REGION Network 162: Reset CV nước Bồn 3 khi không dosing
   RUNG wire#powerrail
      I_Contact( "PLC2_Step_Bon3_Dosing" )
      { S7_GenerateENO := "TRUE" } Move(in := 0.0, out1 => "CV3211_Nuoc_Bon3")
   END_RUNG
   // the same network as SCL:
   IF NOT "PLC2_Step_Bon3_Dosing" THEN "CV3211_Nuoc_Bon3" := 0.0; END_IF;
END_REGION

REGION Network 163: Reset CV nước Bồn 3 khi Stop hoặc Lỗi tổng PLC2
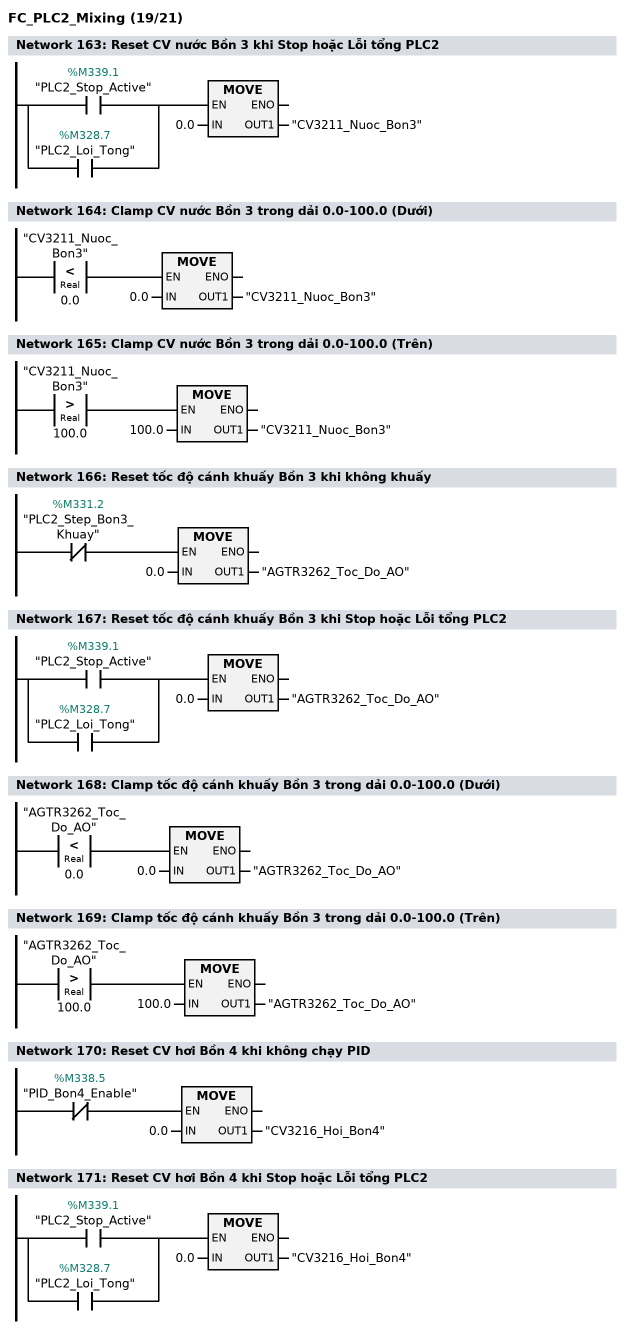
   RUNG wire#powerrail
      Contact( "PLC2_Stop_Active" )
      wire#w1
      { S7_GenerateENO := "TRUE" } Move(in := 0.0, out1 => "CV3211_Nuoc_Bon3")
   END_RUNG
   RUNG wire#powerrail
      Contact( "PLC2_Loi_Tong" )
   END_RUNG wire#w1
   // the same network as SCL:
   IF "PLC2_Stop_Active" OR "PLC2_Loi_Tong" THEN "CV3211_Nuoc_Bon3" := 0.0; END_IF;
END_REGION

REGION Network 164: Clamp CV nước Bồn 3 trong dải 0.0-100.0 (Dưới)
   RUNG wire#powerrail
      { S7_Templates := "SrcType := Real" } LT_Contact(in1 := "CV3211_Nuoc_Bon3", in2 := 0.0)
      { S7_GenerateENO := "TRUE" } Move(in := 0.0, out1 => "CV3211_Nuoc_Bon3")
   END_RUNG
   // the same network as SCL:
   IF "CV3211_Nuoc_Bon3" < 0.0 THEN "CV3211_Nuoc_Bon3" := 0.0; END_IF;
END_REGION

REGION Network 165: Clamp CV nước Bồn 3 trong dải 0.0-100.0 (Trên)
   RUNG wire#powerrail
      { S7_Templates := "SrcType := Real" } GT_Contact(in1 := "CV3211_Nuoc_Bon3", in2 := 100.0)
      { S7_GenerateENO := "TRUE" } Move(in := 100.0, out1 => "CV3211_Nuoc_Bon3")
   END_RUNG
   // the same network as SCL:
   IF "CV3211_Nuoc_Bon3" > 100.0 THEN "CV3211_Nuoc_Bon3" := 100.0; END_IF;
END_REGION

REGION Network 166: Reset tốc độ cánh khuấy Bồn 3 khi không khuấy
   RUNG wire#powerrail
      I_Contact( "PLC2_Step_Bon3_Khuay" )
      { S7_GenerateENO := "TRUE" } Move(in := 0.0, out1 => "AGTR3262_Toc_Do_AO")
   END_RUNG
   // the same network as SCL:
   IF NOT "PLC2_Step_Bon3_Khuay" THEN "AGTR3262_Toc_Do_AO" := 0.0; END_IF;
END_REGION

REGION Network 167: Reset tốc độ cánh khuấy Bồn 3 khi Stop hoặc Lỗi tổng PLC2
   RUNG wire#powerrail
      Contact( "PLC2_Stop_Active" )
      wire#w1
      { S7_GenerateENO := "TRUE" } Move(in := 0.0, out1 => "AGTR3262_Toc_Do_AO")
   END_RUNG
   RUNG wire#powerrail
      Contact( "PLC2_Loi_Tong" )
   END_RUNG wire#w1
   // the same network as SCL:
   IF "PLC2_Stop_Active" OR "PLC2_Loi_Tong" THEN "AGTR3262_Toc_Do_AO" := 0.0; END_IF;
END_REGION

REGION Network 168: Clamp tốc độ cánh khuấy Bồn 3 trong dải 0.0-100.0 (Dưới)
   RUNG wire#powerrail
      { S7_Templates := "SrcType := Real" } LT_Contact(in1 := "AGTR3262_Toc_Do_AO", in2 := 0.0)
      { S7_GenerateENO := "TRUE" } Move(in := 0.0, out1 => "AGTR3262_Toc_Do_AO")
   END_RUNG
   // the same network as SCL:
   IF "AGTR3262_Toc_Do_AO" < 0.0 THEN "AGTR3262_Toc_Do_AO" := 0.0; END_IF;
END_REGION

REGION Network 169: Clamp tốc độ cánh khuấy Bồn 3 trong dải 0.0-100.0 (Trên)
   RUNG wire#powerrail
      { S7_Templates := "SrcType := Real" } GT_Contact(in1 := "AGTR3262_Toc_Do_AO", in2 := 100.0)
      { S7_GenerateENO := "TRUE" } Move(in := 100.0, out1 => "AGTR3262_Toc_Do_AO")
   END_RUNG
   // the same network as SCL:
   IF "AGTR3262_Toc_Do_AO" > 100.0 THEN "AGTR3262_Toc_Do_AO" := 100.0; END_IF;
END_REGION

REGION Network 170: Reset CV hơi Bồn 4 khi không chạy PID
   RUNG wire#powerrail
      I_Contact( "PID_Bon4_Enable" )
      { S7_GenerateENO := "TRUE" } Move(in := 0.0, out1 => "CV3216_Hoi_Bon4")
   END_RUNG
   // the same network as SCL:
   IF NOT "PID_Bon4_Enable" THEN "CV3216_Hoi_Bon4" := 0.0; END_IF;
END_REGION

REGION Network 171: Reset CV hơi Bồn 4 khi Stop hoặc Lỗi tổng PLC2
   RUNG wire#powerrail
      Contact( "PLC2_Stop_Active" )
      wire#w1
      { S7_GenerateENO := "TRUE" } Move(in := 0.0, out1 => "CV3216_Hoi_Bon4")
   END_RUNG
   RUNG wire#powerrail
      Contact( "PLC2_Loi_Tong" )
   END_RUNG wire#w1
   // the same network as SCL:
   IF "PLC2_Stop_Active" OR "PLC2_Loi_Tong" THEN "CV3216_Hoi_Bon4" := 0.0; END_IF;
END_REGION

REGION Network 172: Clamp CV hơi Bồn 4 trong dải 0.0-100.0 (Dưới)
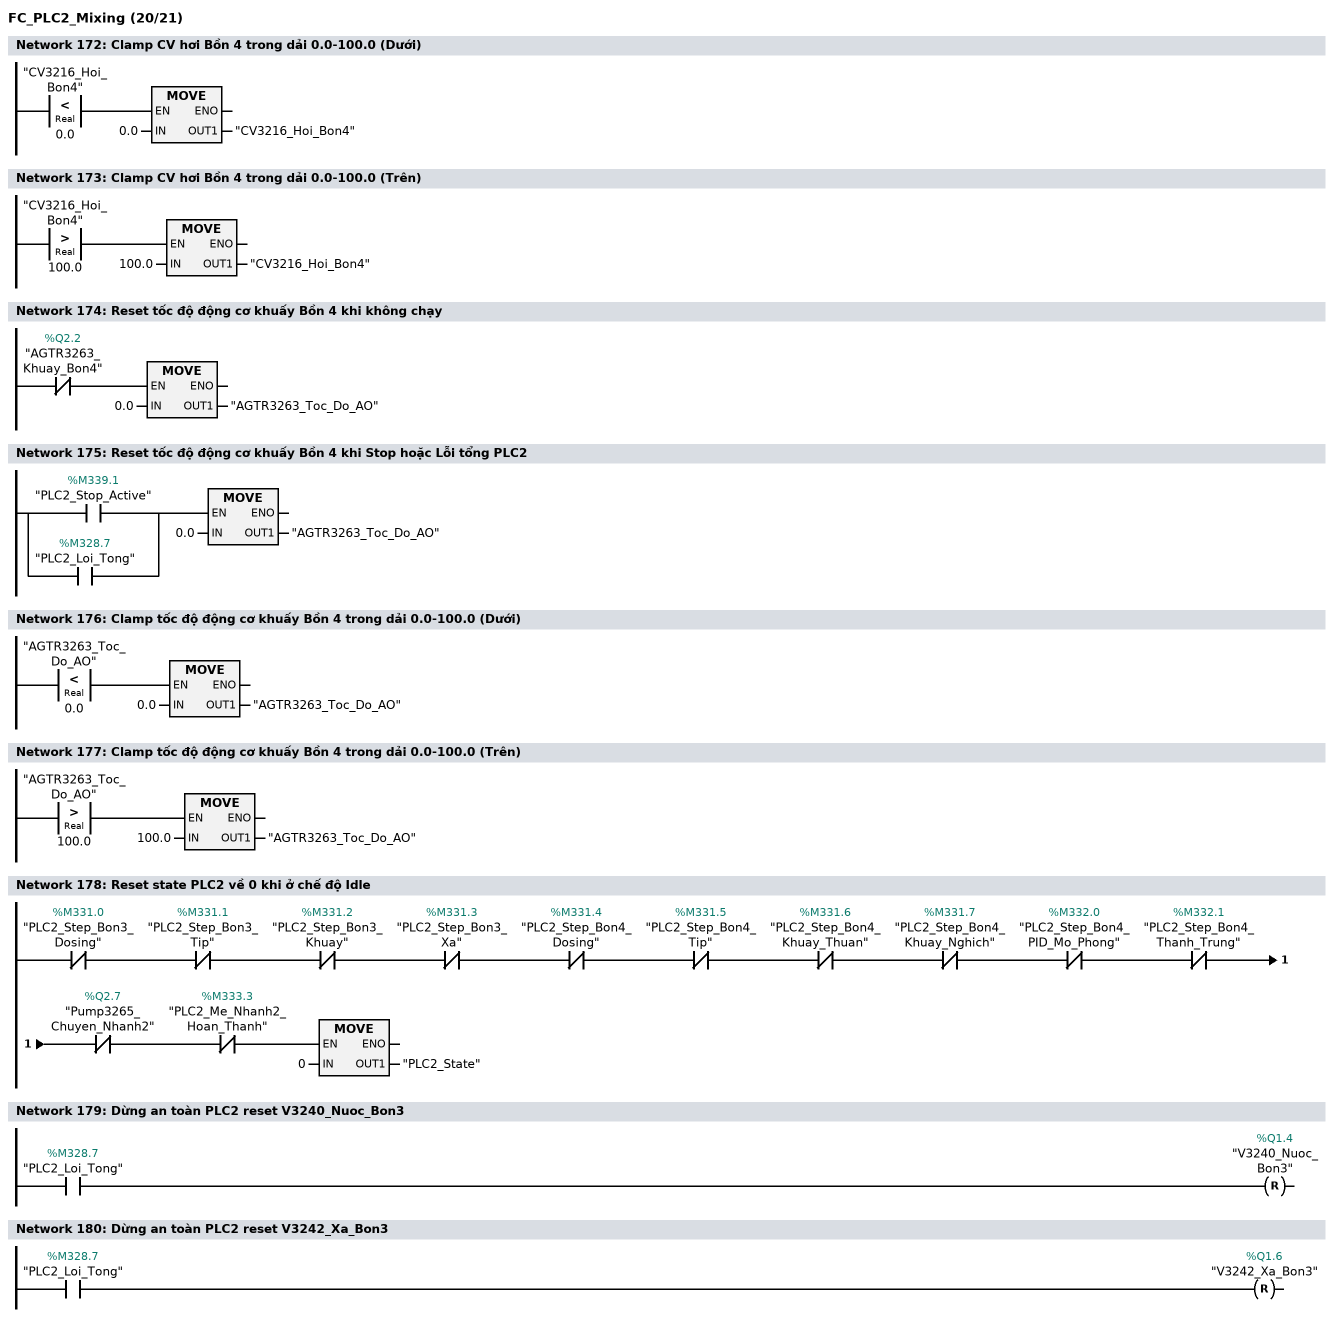
   RUNG wire#powerrail
      { S7_Templates := "SrcType := Real" } LT_Contact(in1 := "CV3216_Hoi_Bon4", in2 := 0.0)
      { S7_GenerateENO := "TRUE" } Move(in := 0.0, out1 => "CV3216_Hoi_Bon4")
   END_RUNG
   // the same network as SCL:
   IF "CV3216_Hoi_Bon4" < 0.0 THEN "CV3216_Hoi_Bon4" := 0.0; END_IF;
END_REGION

REGION Network 173: Clamp CV hơi Bồn 4 trong dải 0.0-100.0 (Trên)
   RUNG wire#powerrail
      { S7_Templates := "SrcType := Real" } GT_Contact(in1 := "CV3216_Hoi_Bon4", in2 := 100.0)
      { S7_GenerateENO := "TRUE" } Move(in := 100.0, out1 => "CV3216_Hoi_Bon4")
   END_RUNG
   // the same network as SCL:
   IF "CV3216_Hoi_Bon4" > 100.0 THEN "CV3216_Hoi_Bon4" := 100.0; END_IF;
END_REGION

REGION Network 174: Reset tốc độ động cơ khuấy Bồn 4 khi không chạy
   RUNG wire#powerrail
      I_Contact( "AGTR3263_Khuay_Bon4" )
      { S7_GenerateENO := "TRUE" } Move(in := 0.0, out1 => "AGTR3263_Toc_Do_AO")
   END_RUNG
   // the same network as SCL:
   IF NOT "AGTR3263_Khuay_Bon4" THEN "AGTR3263_Toc_Do_AO" := 0.0; END_IF;
END_REGION

REGION Network 175: Reset tốc độ động cơ khuấy Bồn 4 khi Stop hoặc Lỗi tổng PLC2
   RUNG wire#powerrail
      Contact( "PLC2_Stop_Active" )
      wire#w1
      { S7_GenerateENO := "TRUE" } Move(in := 0.0, out1 => "AGTR3263_Toc_Do_AO")
   END_RUNG
   RUNG wire#powerrail
      Contact( "PLC2_Loi_Tong" )
   END_RUNG wire#w1
   // the same network as SCL:
   IF "PLC2_Stop_Active" OR "PLC2_Loi_Tong" THEN "AGTR3263_Toc_Do_AO" := 0.0; END_IF;
END_REGION

REGION Network 176: Clamp tốc độ động cơ khuấy Bồn 4 trong dải 0.0-100.0 (Dưới)
   RUNG wire#powerrail
      { S7_Templates := "SrcType := Real" } LT_Contact(in1 := "AGTR3263_Toc_Do_AO", in2 := 0.0)
      { S7_GenerateENO := "TRUE" } Move(in := 0.0, out1 => "AGTR3263_Toc_Do_AO")
   END_RUNG
   // the same network as SCL:
   IF "AGTR3263_Toc_Do_AO" < 0.0 THEN "AGTR3263_Toc_Do_AO" := 0.0; END_IF;
END_REGION

REGION Network 177: Clamp tốc độ động cơ khuấy Bồn 4 trong dải 0.0-100.0 (Trên)
   RUNG wire#powerrail
      { S7_Templates := "SrcType := Real" } GT_Contact(in1 := "AGTR3263_Toc_Do_AO", in2 := 100.0)
      { S7_GenerateENO := "TRUE" } Move(in := 100.0, out1 => "AGTR3263_Toc_Do_AO")
   END_RUNG
   // the same network as SCL:
   IF "AGTR3263_Toc_Do_AO" > 100.0 THEN "AGTR3263_Toc_Do_AO" := 100.0; END_IF;
END_REGION

REGION Network 178: Reset state PLC2 về 0 khi ở chế độ Idle
   RUNG wire#powerrail
      I_Contact( "PLC2_Step_Bon3_Dosing" )
      I_Contact( "PLC2_Step_Bon3_Tip" )
      I_Contact( "PLC2_Step_Bon3_Khuay" )
      I_Contact( "PLC2_Step_Bon3_Xa" )
      I_Contact( "PLC2_Step_Bon4_Dosing" )
      I_Contact( "PLC2_Step_Bon4_Tip" )
      I_Contact( "PLC2_Step_Bon4_Khuay_Thuan" )
      I_Contact( "PLC2_Step_Bon4_Khuay_Nghich" )
      I_Contact( "PLC2_Step_Bon4_PID_Mo_Phong" )
      I_Contact( "PLC2_Step_Bon4_Thanh_Trung" )
      I_Contact( "Pump3265_Chuyen_Nhanh2" )
      I_Contact( "PLC2_Me_Nhanh2_Hoan_Thanh" )
      { S7_GenerateENO := "TRUE" } Move(in := 0, out1 => "PLC2_State")
   END_RUNG
   // the same network as SCL:
   IF NOT "PLC2_Step_Bon3_Dosing" AND NOT "PLC2_Step_Bon3_Tip" AND NOT "PLC2_Step_Bon3_Khuay" AND NOT "PLC2_Step_Bon3_Xa" AND NOT "PLC2_Step_Bon4_Dosing" AND NOT "PLC2_Step_Bon4_Tip" AND NOT "PLC2_Step_Bon4_Khuay_Thuan" AND NOT "PLC2_Step_Bon4_Khuay_Nghich" AND NOT "PLC2_Step_Bon4_PID_Mo_Phong" AND NOT "PLC2_Step_Bon4_Thanh_Trung" AND NOT "Pump3265_Chuyen_Nhanh2" AND NOT "PLC2_Me_Nhanh2_Hoan_Thanh" THEN
       "PLC2_State" := 0;
   END_IF;
END_REGION

REGION Network 179: Dừng an toàn PLC2 reset V3240_Nuoc_Bon3
   RUNG wire#powerrail
      Contact( "PLC2_Loi_Tong" )
      R_Coil( "V3240_Nuoc_Bon3" )
   END_RUNG
   // the same network as SCL:
   IF "PLC2_Loi_Tong" THEN "V3240_Nuoc_Bon3" := FALSE; END_IF;
END_REGION

REGION Network 180: Dừng an toàn PLC2 reset V3242_Xa_Bon3
   RUNG wire#powerrail
      Contact( "PLC2_Loi_Tong" )
      R_Coil( "V3242_Xa_Bon3" )
   END_RUNG
   // the same network as SCL:
   IF "PLC2_Loi_Tong" THEN "V3242_Xa_Bon3" := FALSE; END_IF;
END_REGION

REGION Network 181: Dừng an toàn PLC2 reset V3243_Xa_Bon3
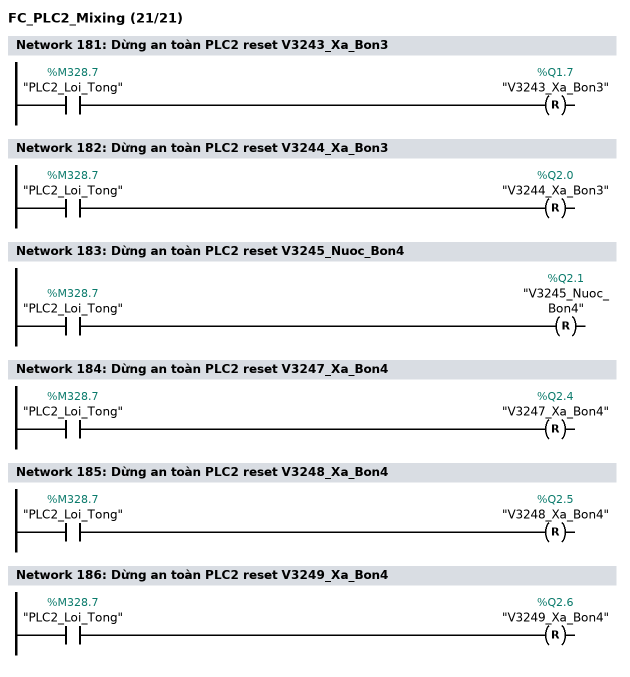
   RUNG wire#powerrail
      Contact( "PLC2_Loi_Tong" )
      R_Coil( "V3243_Xa_Bon3" )
   END_RUNG
   // the same network as SCL:
   IF "PLC2_Loi_Tong" THEN "V3243_Xa_Bon3" := FALSE; END_IF;
END_REGION

REGION Network 182: Dừng an toàn PLC2 reset V3244_Xa_Bon3
   RUNG wire#powerrail
      Contact( "PLC2_Loi_Tong" )
      R_Coil( "V3244_Xa_Bon3" )
   END_RUNG
   // the same network as SCL:
   IF "PLC2_Loi_Tong" THEN "V3244_Xa_Bon3" := FALSE; END_IF;
END_REGION

REGION Network 183: Dừng an toàn PLC2 reset V3245_Nuoc_Bon4
   RUNG wire#powerrail
      Contact( "PLC2_Loi_Tong" )
      R_Coil( "V3245_Nuoc_Bon4" )
   END_RUNG
   // the same network as SCL:
   IF "PLC2_Loi_Tong" THEN "V3245_Nuoc_Bon4" := FALSE; END_IF;
END_REGION

REGION Network 184: Dừng an toàn PLC2 reset V3247_Xa_Bon4
   RUNG wire#powerrail
      Contact( "PLC2_Loi_Tong" )
      R_Coil( "V3247_Xa_Bon4" )
   END_RUNG
   // the same network as SCL:
   IF "PLC2_Loi_Tong" THEN "V3247_Xa_Bon4" := FALSE; END_IF;
END_REGION

REGION Network 185: Dừng an toàn PLC2 reset V3248_Xa_Bon4
   RUNG wire#powerrail
      Contact( "PLC2_Loi_Tong" )
      R_Coil( "V3248_Xa_Bon4" )
   END_RUNG
   // the same network as SCL:
   IF "PLC2_Loi_Tong" THEN "V3248_Xa_Bon4" := FALSE; END_IF;
END_REGION

REGION Network 186: Dừng an toàn PLC2 reset V3249_Xa_Bon4
   RUNG wire#powerrail
      Contact( "PLC2_Loi_Tong" )
      R_Coil( "V3249_Xa_Bon4" )
   END_RUNG
   // the same network as SCL:
   IF "PLC2_Loi_Tong" THEN "V3249_Xa_Bon4" := FALSE; END_IF;
END_REGION
END_FUNCTION

FUNCTION "FC_HMI_Mirror_PLC2" : Void   // FC41, LAD
{ S7_Optimized_Access := 'TRUE' }
VERSION : 0.1
// stored: AutoNumber true, IsIECCheckEnabled false, SetENOAutomatically false, UDAEnableTagReadback false
BEGIN

REGION Network 1: Mirror V3240_Nuoc_Bon3
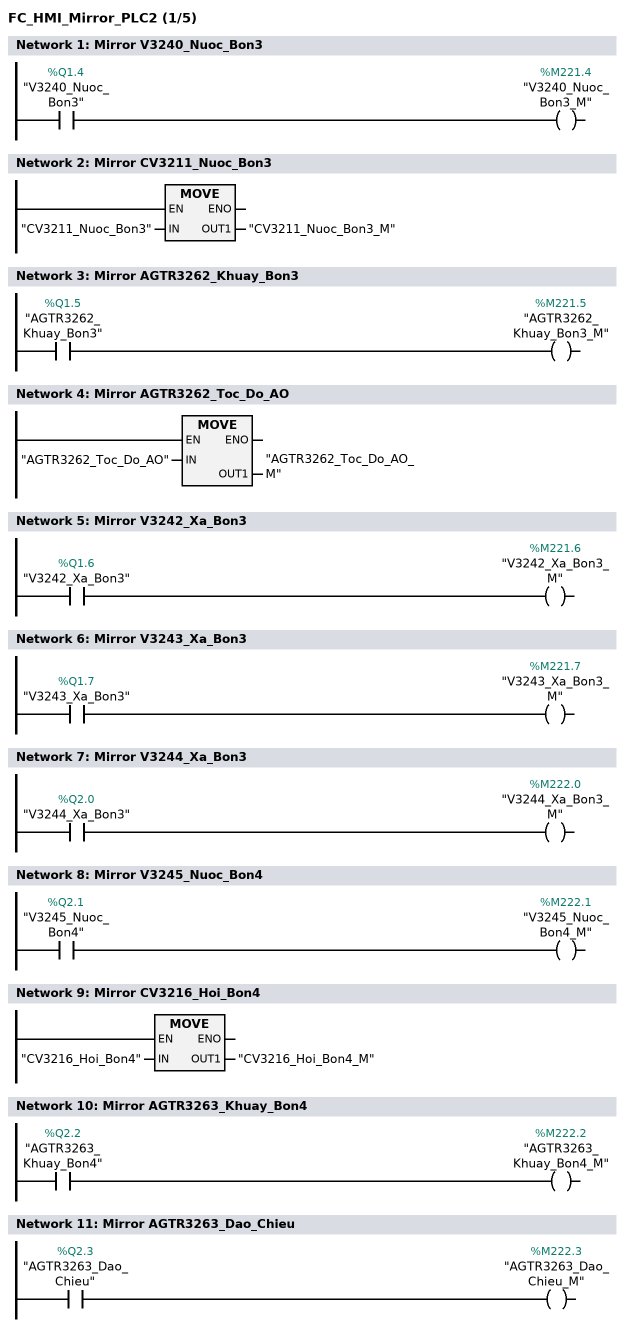
   RUNG wire#powerrail
      Contact( "V3240_Nuoc_Bon3" )
      Coil( "V3240_Nuoc_Bon3_M" )
   END_RUNG
   // the same network as SCL:
   "V3240_Nuoc_Bon3_M" := "V3240_Nuoc_Bon3";
END_REGION

REGION Network 2: Mirror CV3211_Nuoc_Bon3
   RUNG wire#powerrail
      { S7_GenerateENO := "TRUE" } Move(in := "CV3211_Nuoc_Bon3", out1 => "CV3211_Nuoc_Bon3_M")
   END_RUNG
   // the same network as SCL:
   "CV3211_Nuoc_Bon3_M" := "CV3211_Nuoc_Bon3";
END_REGION

REGION Network 3: Mirror AGTR3262_Khuay_Bon3
   RUNG wire#powerrail
      Contact( "AGTR3262_Khuay_Bon3" )
      Coil( "AGTR3262_Khuay_Bon3_M" )
   END_RUNG
   // the same network as SCL:
   "AGTR3262_Khuay_Bon3_M" := "AGTR3262_Khuay_Bon3";
END_REGION

REGION Network 4: Mirror AGTR3262_Toc_Do_AO
   RUNG wire#powerrail
      { S7_GenerateENO := "TRUE" } Move(in := "AGTR3262_Toc_Do_AO", out1 => "AGTR3262_Toc_Do_AO_M")
   END_RUNG
   // the same network as SCL:
   "AGTR3262_Toc_Do_AO_M" := "AGTR3262_Toc_Do_AO";
END_REGION

REGION Network 5: Mirror V3242_Xa_Bon3
   RUNG wire#powerrail
      Contact( "V3242_Xa_Bon3" )
      Coil( "V3242_Xa_Bon3_M" )
   END_RUNG
   // the same network as SCL:
   "V3242_Xa_Bon3_M" := "V3242_Xa_Bon3";
END_REGION

REGION Network 6: Mirror V3243_Xa_Bon3
   RUNG wire#powerrail
      Contact( "V3243_Xa_Bon3" )
      Coil( "V3243_Xa_Bon3_M" )
   END_RUNG
   // the same network as SCL:
   "V3243_Xa_Bon3_M" := "V3243_Xa_Bon3";
END_REGION

REGION Network 7: Mirror V3244_Xa_Bon3
   RUNG wire#powerrail
      Contact( "V3244_Xa_Bon3" )
      Coil( "V3244_Xa_Bon3_M" )
   END_RUNG
   // the same network as SCL:
   "V3244_Xa_Bon3_M" := "V3244_Xa_Bon3";
END_REGION

REGION Network 8: Mirror V3245_Nuoc_Bon4
   RUNG wire#powerrail
      Contact( "V3245_Nuoc_Bon4" )
      Coil( "V3245_Nuoc_Bon4_M" )
   END_RUNG
   // the same network as SCL:
   "V3245_Nuoc_Bon4_M" := "V3245_Nuoc_Bon4";
END_REGION

REGION Network 9: Mirror CV3216_Hoi_Bon4
   RUNG wire#powerrail
      { S7_GenerateENO := "TRUE" } Move(in := "CV3216_Hoi_Bon4", out1 => "CV3216_Hoi_Bon4_M")
   END_RUNG
   // the same network as SCL:
   "CV3216_Hoi_Bon4_M" := "CV3216_Hoi_Bon4";
END_REGION

REGION Network 10: Mirror AGTR3263_Khuay_Bon4
   RUNG wire#powerrail
      Contact( "AGTR3263_Khuay_Bon4" )
      Coil( "AGTR3263_Khuay_Bon4_M" )
   END_RUNG
   // the same network as SCL:
   "AGTR3263_Khuay_Bon4_M" := "AGTR3263_Khuay_Bon4";
END_REGION

REGION Network 11: Mirror AGTR3263_Dao_Chieu
   RUNG wire#powerrail
      Contact( "AGTR3263_Dao_Chieu" )
      Coil( "AGTR3263_Dao_Chieu_M" )
   END_RUNG
   // the same network as SCL:
   "AGTR3263_Dao_Chieu_M" := "AGTR3263_Dao_Chieu";
END_REGION

REGION Network 12: Mirror AGTR3263_Toc_Do_AO
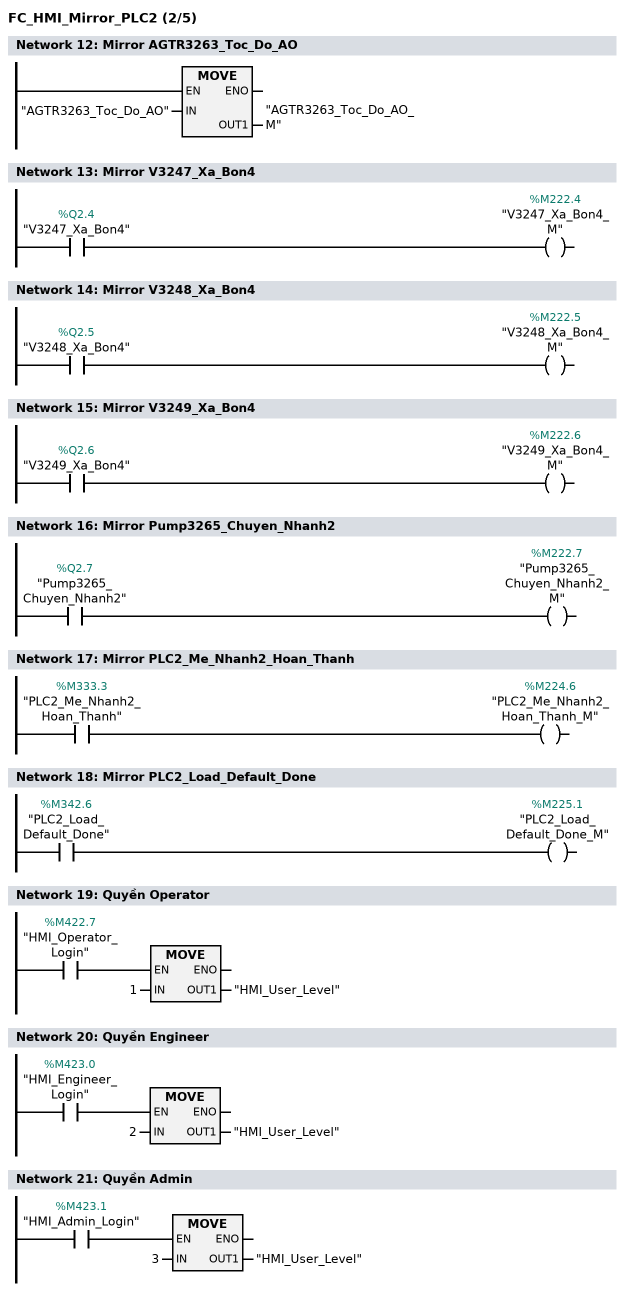
   RUNG wire#powerrail
      { S7_GenerateENO := "TRUE" } Move(in := "AGTR3263_Toc_Do_AO", out1 => "AGTR3263_Toc_Do_AO_M")
   END_RUNG
   // the same network as SCL:
   "AGTR3263_Toc_Do_AO_M" := "AGTR3263_Toc_Do_AO";
END_REGION

REGION Network 13: Mirror V3247_Xa_Bon4
   RUNG wire#powerrail
      Contact( "V3247_Xa_Bon4" )
      Coil( "V3247_Xa_Bon4_M" )
   END_RUNG
   // the same network as SCL:
   "V3247_Xa_Bon4_M" := "V3247_Xa_Bon4";
END_REGION

REGION Network 14: Mirror V3248_Xa_Bon4
   RUNG wire#powerrail
      Contact( "V3248_Xa_Bon4" )
      Coil( "V3248_Xa_Bon4_M" )
   END_RUNG
   // the same network as SCL:
   "V3248_Xa_Bon4_M" := "V3248_Xa_Bon4";
END_REGION

REGION Network 15: Mirror V3249_Xa_Bon4
   RUNG wire#powerrail
      Contact( "V3249_Xa_Bon4" )
      Coil( "V3249_Xa_Bon4_M" )
   END_RUNG
   // the same network as SCL:
   "V3249_Xa_Bon4_M" := "V3249_Xa_Bon4";
END_REGION

REGION Network 16: Mirror Pump3265_Chuyen_Nhanh2
   RUNG wire#powerrail
      Contact( "Pump3265_Chuyen_Nhanh2" )
      Coil( "Pump3265_Chuyen_Nhanh2_M" )
   END_RUNG
   // the same network as SCL:
   "Pump3265_Chuyen_Nhanh2_M" := "Pump3265_Chuyen_Nhanh2";
END_REGION

REGION Network 17: Mirror PLC2_Me_Nhanh2_Hoan_Thanh
   RUNG wire#powerrail
      Contact( "PLC2_Me_Nhanh2_Hoan_Thanh" )
      Coil( "PLC2_Me_Nhanh2_Hoan_Thanh_M" )
   END_RUNG
   // the same network as SCL:
   "PLC2_Me_Nhanh2_Hoan_Thanh_M" := "PLC2_Me_Nhanh2_Hoan_Thanh";
END_REGION

REGION Network 18: Mirror PLC2_Load_Default_Done
   RUNG wire#powerrail
      Contact( "PLC2_Load_Default_Done" )
      Coil( "PLC2_Load_Default_Done_M" )
   END_RUNG
   // the same network as SCL:
   "PLC2_Load_Default_Done_M" := "PLC2_Load_Default_Done";
END_REGION

REGION Network 19: Quyền Operator
   RUNG wire#powerrail
      Contact( "HMI_Operator_Login" )
      { S7_GenerateENO := "TRUE" } Move(in := 1, out1 => "HMI_User_Level")
   END_RUNG
   // the same network as SCL:
   IF "HMI_Operator_Login" THEN "HMI_User_Level" := 1; END_IF;
END_REGION

REGION Network 20: Quyền Engineer
   RUNG wire#powerrail
      Contact( "HMI_Engineer_Login" )
      { S7_GenerateENO := "TRUE" } Move(in := 2, out1 => "HMI_User_Level")
   END_RUNG
   // the same network as SCL:
   IF "HMI_Engineer_Login" THEN "HMI_User_Level" := 2; END_IF;
END_REGION

REGION Network 21: Quyền Admin
   RUNG wire#powerrail
      Contact( "HMI_Admin_Login" )
      { S7_GenerateENO := "TRUE" } Move(in := 3, out1 => "HMI_User_Level")
   END_RUNG
   // the same network as SCL:
   IF "HMI_Admin_Login" THEN "HMI_User_Level" := 3; END_IF;
END_REGION

REGION Network 22: Cho phép sửa thông số Engineer
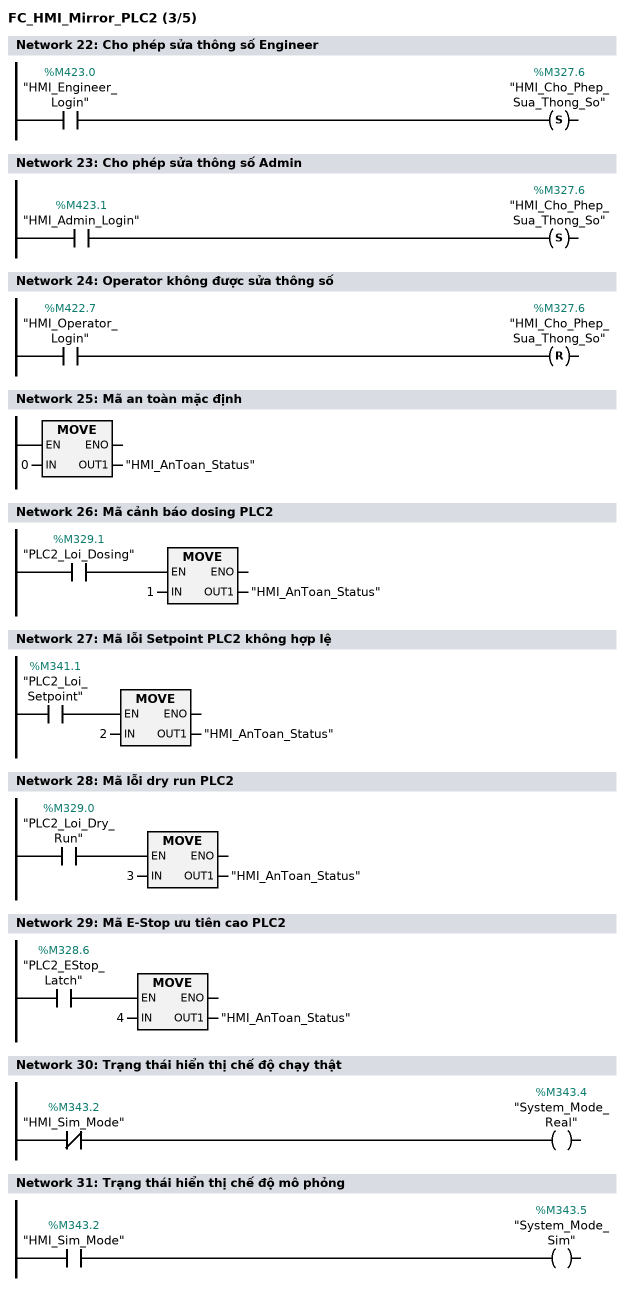
   RUNG wire#powerrail
      Contact( "HMI_Engineer_Login" )
      S_Coil( "HMI_Cho_Phep_Sua_Thong_So" )
   END_RUNG
   // the same network as SCL:
   IF "HMI_Engineer_Login" THEN "HMI_Cho_Phep_Sua_Thong_So" := TRUE; END_IF;
END_REGION

REGION Network 23: Cho phép sửa thông số Admin
   RUNG wire#powerrail
      Contact( "HMI_Admin_Login" )
      S_Coil( "HMI_Cho_Phep_Sua_Thong_So" )
   END_RUNG
   // the same network as SCL:
   IF "HMI_Admin_Login" THEN "HMI_Cho_Phep_Sua_Thong_So" := TRUE; END_IF;
END_REGION

REGION Network 24: Operator không được sửa thông số
   RUNG wire#powerrail
      Contact( "HMI_Operator_Login" )
      R_Coil( "HMI_Cho_Phep_Sua_Thong_So" )
   END_RUNG
   // the same network as SCL:
   IF "HMI_Operator_Login" THEN "HMI_Cho_Phep_Sua_Thong_So" := FALSE; END_IF;
END_REGION

REGION Network 25: Mã an toàn mặc định
   RUNG wire#powerrail
      { S7_GenerateENO := "TRUE" } Move(in := 0, out1 => "HMI_AnToan_Status")
   END_RUNG
   // the same network as SCL:
   "HMI_AnToan_Status" := 0;
END_REGION

REGION Network 26: Mã cảnh báo dosing PLC2
   RUNG wire#powerrail
      Contact( "PLC2_Loi_Dosing" )
      { S7_GenerateENO := "TRUE" } Move(in := 1, out1 => "HMI_AnToan_Status")
   END_RUNG
   // the same network as SCL:
   IF "PLC2_Loi_Dosing" THEN "HMI_AnToan_Status" := 1; END_IF;
END_REGION

REGION Network 27: Mã lỗi Setpoint PLC2 không hợp lệ
   RUNG wire#powerrail
      Contact( "PLC2_Loi_Setpoint" )
      { S7_GenerateENO := "TRUE" } Move(in := 2, out1 => "HMI_AnToan_Status")
   END_RUNG
   // the same network as SCL:
   IF "PLC2_Loi_Setpoint" THEN "HMI_AnToan_Status" := 2; END_IF;
END_REGION

REGION Network 28: Mã lỗi dry run PLC2
   RUNG wire#powerrail
      Contact( "PLC2_Loi_Dry_Run" )
      { S7_GenerateENO := "TRUE" } Move(in := 3, out1 => "HMI_AnToan_Status")
   END_RUNG
   // the same network as SCL:
   IF "PLC2_Loi_Dry_Run" THEN "HMI_AnToan_Status" := 3; END_IF;
END_REGION

REGION Network 29: Mã E-Stop ưu tiên cao PLC2
   RUNG wire#powerrail
      Contact( "PLC2_EStop_Latch" )
      { S7_GenerateENO := "TRUE" } Move(in := 4, out1 => "HMI_AnToan_Status")
   END_RUNG
   // the same network as SCL:
   IF "PLC2_EStop_Latch" THEN "HMI_AnToan_Status" := 4; END_IF;
END_REGION

REGION Network 30: Trạng thái hiển thị chế độ chạy thật
   RUNG wire#powerrail
      I_Contact( "HMI_Sim_Mode" )
      Coil( "System_Mode_Real" )
   END_RUNG
   // the same network as SCL:
   "System_Mode_Real" := NOT "HMI_Sim_Mode";
END_REGION

REGION Network 31: Trạng thái hiển thị chế độ mô phỏng
   RUNG wire#powerrail
      Contact( "HMI_Sim_Mode" )
      Coil( "System_Mode_Sim" )
   END_RUNG
   // the same network as SCL:
   "System_Mode_Sim" := "HMI_Sim_Mode";
END_REGION

REGION Network 32: Cảnh báo chế độ mô phỏng HMI active
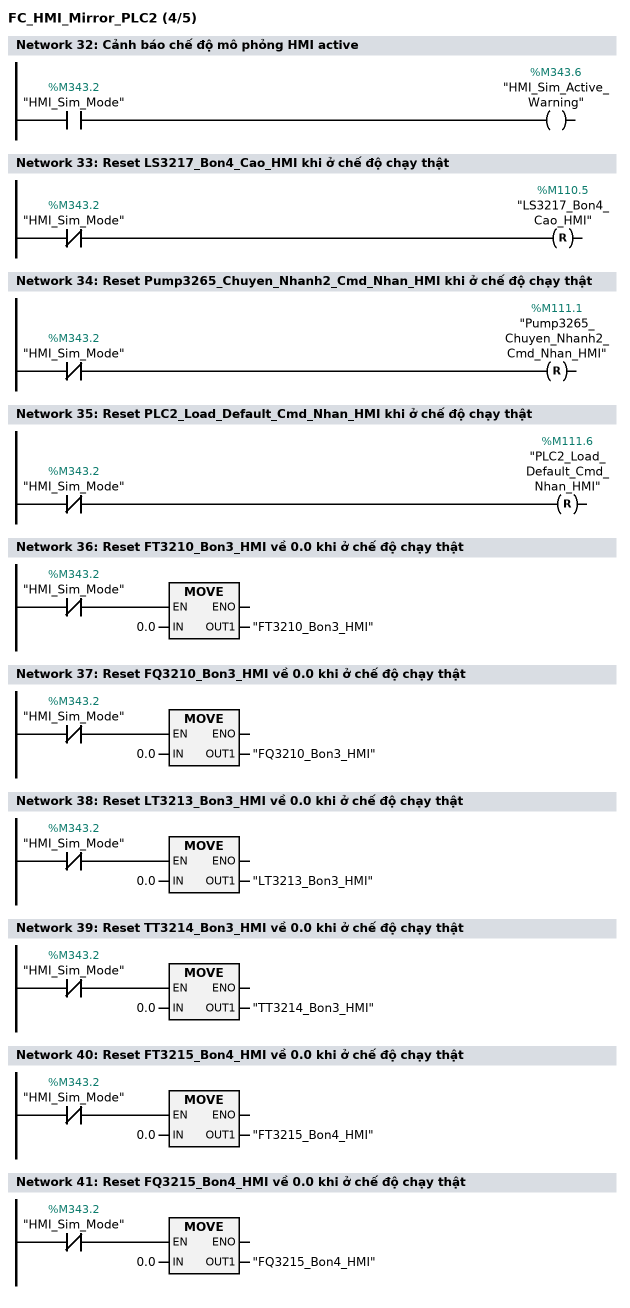
   RUNG wire#powerrail
      Contact( "HMI_Sim_Mode" )
      Coil( "HMI_Sim_Active_Warning" )
   END_RUNG
   // the same network as SCL:
   "HMI_Sim_Active_Warning" := "HMI_Sim_Mode";
END_REGION

REGION Network 33: Reset LS3217_Bon4_Cao_HMI khi ở chế độ chạy thật
   RUNG wire#powerrail
      I_Contact( "HMI_Sim_Mode" )
      R_Coil( "LS3217_Bon4_Cao_HMI" )
   END_RUNG
   // the same network as SCL:
   IF NOT "HMI_Sim_Mode" THEN "LS3217_Bon4_Cao_HMI" := FALSE; END_IF;
END_REGION

REGION Network 34: Reset Pump3265_Chuyen_Nhanh2_Cmd_Nhan_HMI khi ở chế độ chạy thật
   RUNG wire#powerrail
      I_Contact( "HMI_Sim_Mode" )
      R_Coil( "Pump3265_Chuyen_Nhanh2_Cmd_Nhan_HMI" )
   END_RUNG
   // the same network as SCL:
   IF NOT "HMI_Sim_Mode" THEN "Pump3265_Chuyen_Nhanh2_Cmd_Nhan_HMI" := FALSE; END_IF;
END_REGION

REGION Network 35: Reset PLC2_Load_Default_Cmd_Nhan_HMI khi ở chế độ chạy thật
   RUNG wire#powerrail
      I_Contact( "HMI_Sim_Mode" )
      R_Coil( "PLC2_Load_Default_Cmd_Nhan_HMI" )
   END_RUNG
   // the same network as SCL:
   IF NOT "HMI_Sim_Mode" THEN "PLC2_Load_Default_Cmd_Nhan_HMI" := FALSE; END_IF;
END_REGION

REGION Network 36: Reset FT3210_Bon3_HMI về 0.0 khi ở chế độ chạy thật
   RUNG wire#powerrail
      I_Contact( "HMI_Sim_Mode" )
      { S7_GenerateENO := "TRUE" } Move(in := 0.0, out1 => "FT3210_Bon3_HMI")
   END_RUNG
   // the same network as SCL:
   IF NOT "HMI_Sim_Mode" THEN "FT3210_Bon3_HMI" := 0.0; END_IF;
END_REGION

REGION Network 37: Reset FQ3210_Bon3_HMI về 0.0 khi ở chế độ chạy thật
   RUNG wire#powerrail
      I_Contact( "HMI_Sim_Mode" )
      { S7_GenerateENO := "TRUE" } Move(in := 0.0, out1 => "FQ3210_Bon3_HMI")
   END_RUNG
   // the same network as SCL:
   IF NOT "HMI_Sim_Mode" THEN "FQ3210_Bon3_HMI" := 0.0; END_IF;
END_REGION

REGION Network 38: Reset LT3213_Bon3_HMI về 0.0 khi ở chế độ chạy thật
   RUNG wire#powerrail
      I_Contact( "HMI_Sim_Mode" )
      { S7_GenerateENO := "TRUE" } Move(in := 0.0, out1 => "LT3213_Bon3_HMI")
   END_RUNG
   // the same network as SCL:
   IF NOT "HMI_Sim_Mode" THEN "LT3213_Bon3_HMI" := 0.0; END_IF;
END_REGION

REGION Network 39: Reset TT3214_Bon3_HMI về 0.0 khi ở chế độ chạy thật
   RUNG wire#powerrail
      I_Contact( "HMI_Sim_Mode" )
      { S7_GenerateENO := "TRUE" } Move(in := 0.0, out1 => "TT3214_Bon3_HMI")
   END_RUNG
   // the same network as SCL:
   IF NOT "HMI_Sim_Mode" THEN "TT3214_Bon3_HMI" := 0.0; END_IF;
END_REGION

REGION Network 40: Reset FT3215_Bon4_HMI về 0.0 khi ở chế độ chạy thật
   RUNG wire#powerrail
      I_Contact( "HMI_Sim_Mode" )
      { S7_GenerateENO := "TRUE" } Move(in := 0.0, out1 => "FT3215_Bon4_HMI")
   END_RUNG
   // the same network as SCL:
   IF NOT "HMI_Sim_Mode" THEN "FT3215_Bon4_HMI" := 0.0; END_IF;
END_REGION

REGION Network 41: Reset FQ3215_Bon4_HMI về 0.0 khi ở chế độ chạy thật
   RUNG wire#powerrail
      I_Contact( "HMI_Sim_Mode" )
      { S7_GenerateENO := "TRUE" } Move(in := 0.0, out1 => "FQ3215_Bon4_HMI")
   END_RUNG
   // the same network as SCL:
   IF NOT "HMI_Sim_Mode" THEN "FQ3215_Bon4_HMI" := 0.0; END_IF;
END_REGION

REGION Network 42: Reset LT3218_Bon4_HMI về 0.0 khi ở chế độ chạy thật
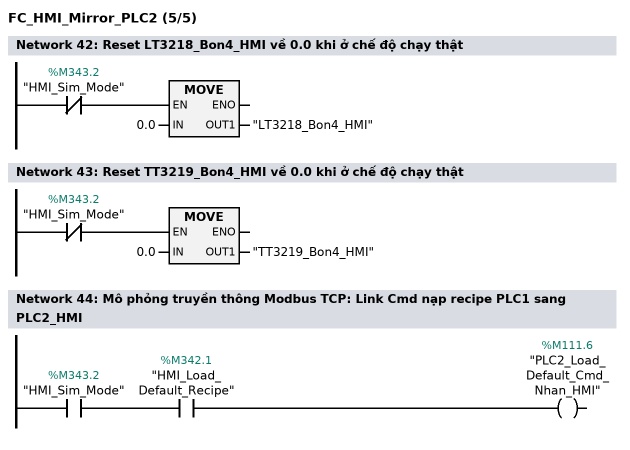
   RUNG wire#powerrail
      I_Contact( "HMI_Sim_Mode" )
      { S7_GenerateENO := "TRUE" } Move(in := 0.0, out1 => "LT3218_Bon4_HMI")
   END_RUNG
   // the same network as SCL:
   IF NOT "HMI_Sim_Mode" THEN "LT3218_Bon4_HMI" := 0.0; END_IF;
END_REGION

REGION Network 43: Reset TT3219_Bon4_HMI về 0.0 khi ở chế độ chạy thật
   RUNG wire#powerrail
      I_Contact( "HMI_Sim_Mode" )
      { S7_GenerateENO := "TRUE" } Move(in := 0.0, out1 => "TT3219_Bon4_HMI")
   END_RUNG
   // the same network as SCL:
   IF NOT "HMI_Sim_Mode" THEN "TT3219_Bon4_HMI" := 0.0; END_IF;
END_REGION

REGION Network 44: Mô phỏng truyền thông Modbus TCP: Link Cmd nạp recipe PLC1 sang PLC2_HMI
   RUNG wire#powerrail
      Contact( "HMI_Sim_Mode" )
      Contact( "HMI_Load_Default_Recipe" )
      Coil( "PLC2_Load_Default_Cmd_Nhan_HMI" )
   END_RUNG
   // the same network as SCL:
   "PLC2_Load_Default_Cmd_Nhan_HMI" := "HMI_Sim_Mode" AND "HMI_Load_Default_Recipe";
END_REGION
END_FUNCTION

ORGANIZATION_BLOCK "OB31_PID_PLC2_Bon4"   // OB31, LAD, CyclicInterrupt
{ S7_Optimized_Access := 'TRUE' }
VERSION : 0.1
// stored: AutoNumber true, IsIECCheckEnabled false, SetENOAutomatically false
   VAR_INPUT
      Initial_Call : Bool;   // Initial call of this OB
      Event_Count : Int;   // Events discarded
   END_VAR
BEGIN

REGION Network 1: Initialize PID Bon 4 Kp parameter
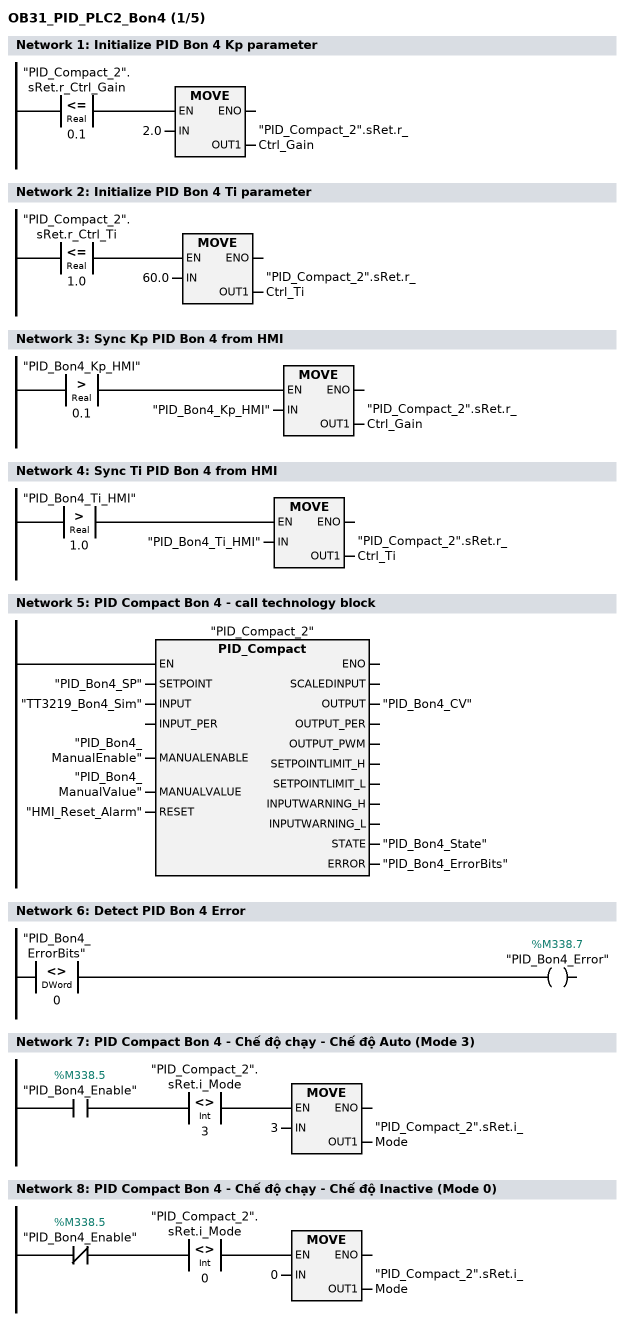
   RUNG wire#powerrail
      { S7_Templates := "SrcType := Real" } LE_Contact(in1 := "PID_Compact_2".sRet.r_Ctrl_Gain, in2 := 0.1)
      { S7_GenerateENO := "TRUE" } Move(in := 2.0, out1 => "PID_Compact_2".sRet.r_Ctrl_Gain)
   END_RUNG
   // the same network as SCL:
   IF "PID_Compact_2".sRet.r_Ctrl_Gain <= 0.1 THEN "PID_Compact_2".sRet.r_Ctrl_Gain := 2.0; END_IF;
END_REGION

REGION Network 2: Initialize PID Bon 4 Ti parameter
   RUNG wire#powerrail
      { S7_Templates := "SrcType := Real" } LE_Contact(in1 := "PID_Compact_2".sRet.r_Ctrl_Ti, in2 := 1.0)
      { S7_GenerateENO := "TRUE" } Move(in := 60.0, out1 => "PID_Compact_2".sRet.r_Ctrl_Ti)
   END_RUNG
   // the same network as SCL:
   IF "PID_Compact_2".sRet.r_Ctrl_Ti <= 1.0 THEN "PID_Compact_2".sRet.r_Ctrl_Ti := 60.0; END_IF;
END_REGION

REGION Network 3: Sync Kp PID Bon 4 from HMI
   RUNG wire#powerrail
      { S7_Templates := "SrcType := Real" } GT_Contact(in1 := "PID_Bon4_Kp_HMI", in2 := 0.1)
      { S7_GenerateENO := "TRUE" } Move(in := "PID_Bon4_Kp_HMI", out1 => "PID_Compact_2".sRet.r_Ctrl_Gain)
   END_RUNG
   // the same network as SCL:
   IF "PID_Bon4_Kp_HMI" > 0.1 THEN "PID_Compact_2".sRet.r_Ctrl_Gain := "PID_Bon4_Kp_HMI"; END_IF;
END_REGION

REGION Network 4: Sync Ti PID Bon 4 from HMI
   RUNG wire#powerrail
      { S7_Templates := "SrcType := Real" } GT_Contact(in1 := "PID_Bon4_Ti_HMI", in2 := 1.0)
      { S7_GenerateENO := "TRUE" } Move(in := "PID_Bon4_Ti_HMI", out1 => "PID_Compact_2".sRet.r_Ctrl_Ti)
   END_RUNG
   // the same network as SCL:
   IF "PID_Bon4_Ti_HMI" > 1.0 THEN "PID_Compact_2".sRet.r_Ctrl_Ti := "PID_Bon4_Ti_HMI"; END_IF;
END_REGION

REGION Network 5: PID Compact Bon 4 - call technology block
   RUNG wire#powerrail
      "PID_Compact_2".PID_Compact(Setpoint := "PID_Bon4_SP", Input := "TT3219_Bon4_Sim", Input_PER :=, ManualEnable := "PID_Bon4_ManualEnable", ManualValue := "PID_Bon4_ManualValue", Reset := "HMI_Reset_Alarm", ScaledInput =>, Output => "PID_Bon4_CV", Output_PER =>, Output_PWM =>, SetpointLimit_H =>, SetpointLimit_L =>, InputWarning_H =>, InputWarning_L =>, State => "PID_Bon4_State", Error => "PID_Bon4_ErrorBits")
   END_RUNG
   // the same network as SCL:
   "PID_Compact_2"(Setpoint := "PID_Bon4_SP",   // PID_Compact
                   Input := "TT3219_Bon4_Sim",
                   ManualEnable := "PID_Bon4_ManualEnable",
                   ManualValue := "PID_Bon4_ManualValue",
                   Reset := "HMI_Reset_Alarm",
                   Output => "PID_Bon4_CV",
                   State => "PID_Bon4_State",
                   Error => "PID_Bon4_ErrorBits");
END_REGION

REGION Network 6: Detect PID Bon 4 Error
   RUNG wire#powerrail
      { S7_Templates := "SrcType := DWord" } NE_Contact(in1 := "PID_Bon4_ErrorBits", in2 := 0)
      Coil( "PID_Bon4_Error" )
   END_RUNG
   // the same network as SCL:
   "PID_Bon4_Error" := "PID_Bon4_ErrorBits" <> 0;
END_REGION

REGION Network 7: PID Compact Bon 4 - Chế độ chạy - Chế độ Auto (Mode 3)
   RUNG wire#powerrail
      Contact( "PID_Bon4_Enable" )
      { S7_Templates := "SrcType := Int" } NE_Contact(in1 := "PID_Compact_2".sRet.i_Mode, in2 := 3)
      { S7_GenerateENO := "TRUE" } Move(in := 3, out1 => "PID_Compact_2".sRet.i_Mode)
   END_RUNG
   // the same network as SCL:
   IF "PID_Bon4_Enable" AND ("PID_Compact_2".sRet.i_Mode <> 3) THEN "PID_Compact_2".sRet.i_Mode := 3; END_IF;
END_REGION

REGION Network 8: PID Compact Bon 4 - Chế độ chạy - Chế độ Inactive (Mode 0)
   RUNG wire#powerrail
      I_Contact( "PID_Bon4_Enable" )
      { S7_Templates := "SrcType := Int" } NE_Contact(in1 := "PID_Compact_2".sRet.i_Mode, in2 := 0)
      { S7_GenerateENO := "TRUE" } Move(in := 0, out1 => "PID_Compact_2".sRet.i_Mode)
   END_RUNG
   // the same network as SCL:
   IF NOT "PID_Bon4_Enable" AND ("PID_Compact_2".sRet.i_Mode <> 0) THEN
       "PID_Compact_2".sRet.i_Mode := 0;
   END_IF;
END_REGION

REGION Network 9: Move PID Bon 4 CV to simulated heat valve
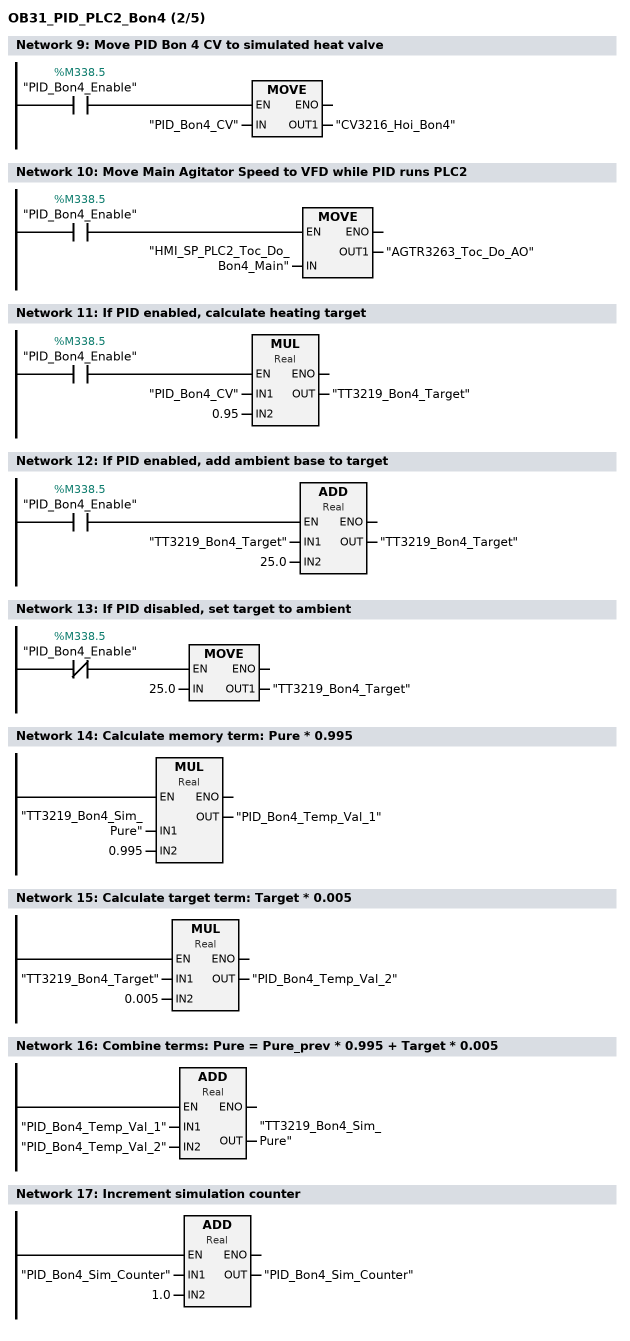
   RUNG wire#powerrail
      Contact( "PID_Bon4_Enable" )
      { S7_GenerateENO := "TRUE" } Move(in := "PID_Bon4_CV", out1 => "CV3216_Hoi_Bon4")
   END_RUNG
   // the same network as SCL:
   IF "PID_Bon4_Enable" THEN "CV3216_Hoi_Bon4" := "PID_Bon4_CV"; END_IF;
END_REGION

REGION Network 10: Move Main Agitator Speed to VFD while PID runs PLC2
   RUNG wire#powerrail
      Contact( "PID_Bon4_Enable" )
      { S7_GenerateENO := "TRUE" } Move(in := "HMI_SP_PLC2_Toc_Do_Bon4_Main", out1 => "AGTR3263_Toc_Do_AO")
   END_RUNG
   // the same network as SCL:
   IF "PID_Bon4_Enable" THEN "AGTR3263_Toc_Do_AO" := "HMI_SP_PLC2_Toc_Do_Bon4_Main"; END_IF;
END_REGION

REGION Network 11: If PID enabled, calculate heating target
   RUNG wire#powerrail
      Contact( "PID_Bon4_Enable" )
      { S7_Templates := "SrcType := Real"; S7_GenerateENO := "TRUE" } Mul(in1 := "PID_Bon4_CV", in2 := 0.95, out => "TT3219_Bon4_Target")
   END_RUNG
   // the same network as SCL:
   IF "PID_Bon4_Enable" THEN "TT3219_Bon4_Target" := "PID_Bon4_CV" * 0.95; END_IF;
END_REGION

REGION Network 12: If PID enabled, add ambient base to target
   RUNG wire#powerrail
      Contact( "PID_Bon4_Enable" )
      { S7_Templates := "SrcType := Real"; S7_GenerateENO := "TRUE" } Add(in1 := "TT3219_Bon4_Target", in2 := 25.0, out => "TT3219_Bon4_Target")
   END_RUNG
   // the same network as SCL:
   IF "PID_Bon4_Enable" THEN "TT3219_Bon4_Target" := "TT3219_Bon4_Target" + 25.0; END_IF;
END_REGION

REGION Network 13: If PID disabled, set target to ambient
   RUNG wire#powerrail
      I_Contact( "PID_Bon4_Enable" )
      { S7_GenerateENO := "TRUE" } Move(in := 25.0, out1 => "TT3219_Bon4_Target")
   END_RUNG
   // the same network as SCL:
   IF NOT "PID_Bon4_Enable" THEN "TT3219_Bon4_Target" := 25.0; END_IF;
END_REGION

REGION Network 14: Calculate memory term: Pure * 0.995
   RUNG wire#powerrail
      { S7_Templates := "SrcType := Real"; S7_GenerateENO := "TRUE" } Mul(in1 := "TT3219_Bon4_Sim_Pure", in2 := 0.995, out => "PID_Bon4_Temp_Val_1")
   END_RUNG
   // the same network as SCL:
   "PID_Bon4_Temp_Val_1" := "TT3219_Bon4_Sim_Pure" * 0.995;
END_REGION

REGION Network 15: Calculate target term: Target * 0.005
   RUNG wire#powerrail
      { S7_Templates := "SrcType := Real"; S7_GenerateENO := "TRUE" } Mul(in1 := "TT3219_Bon4_Target", in2 := 0.005, out => "PID_Bon4_Temp_Val_2")
   END_RUNG
   // the same network as SCL:
   "PID_Bon4_Temp_Val_2" := "TT3219_Bon4_Target" * 0.005;
END_REGION

REGION Network 16: Combine terms: Pure = Pure_prev * 0.995 + Target * 0.005
   RUNG wire#powerrail
      { S7_Templates := "SrcType := Real"; S7_GenerateENO := "TRUE" } Add(in1 := "PID_Bon4_Temp_Val_1", in2 := "PID_Bon4_Temp_Val_2", out => "TT3219_Bon4_Sim_Pure")
   END_RUNG
   // the same network as SCL:
   "TT3219_Bon4_Sim_Pure" := "PID_Bon4_Temp_Val_1" + "PID_Bon4_Temp_Val_2";
END_REGION

REGION Network 17: Increment simulation counter
   RUNG wire#powerrail
      { S7_Templates := "SrcType := Real"; S7_GenerateENO := "TRUE" } Add(in1 := "PID_Bon4_Sim_Counter", in2 := 1.0, out => "PID_Bon4_Sim_Counter")
   END_RUNG
   // the same network as SCL:
   "PID_Bon4_Sim_Counter" := "PID_Bon4_Sim_Counter" + 1.0;
END_REGION

REGION Network 18: Reset simulation counter at 1000
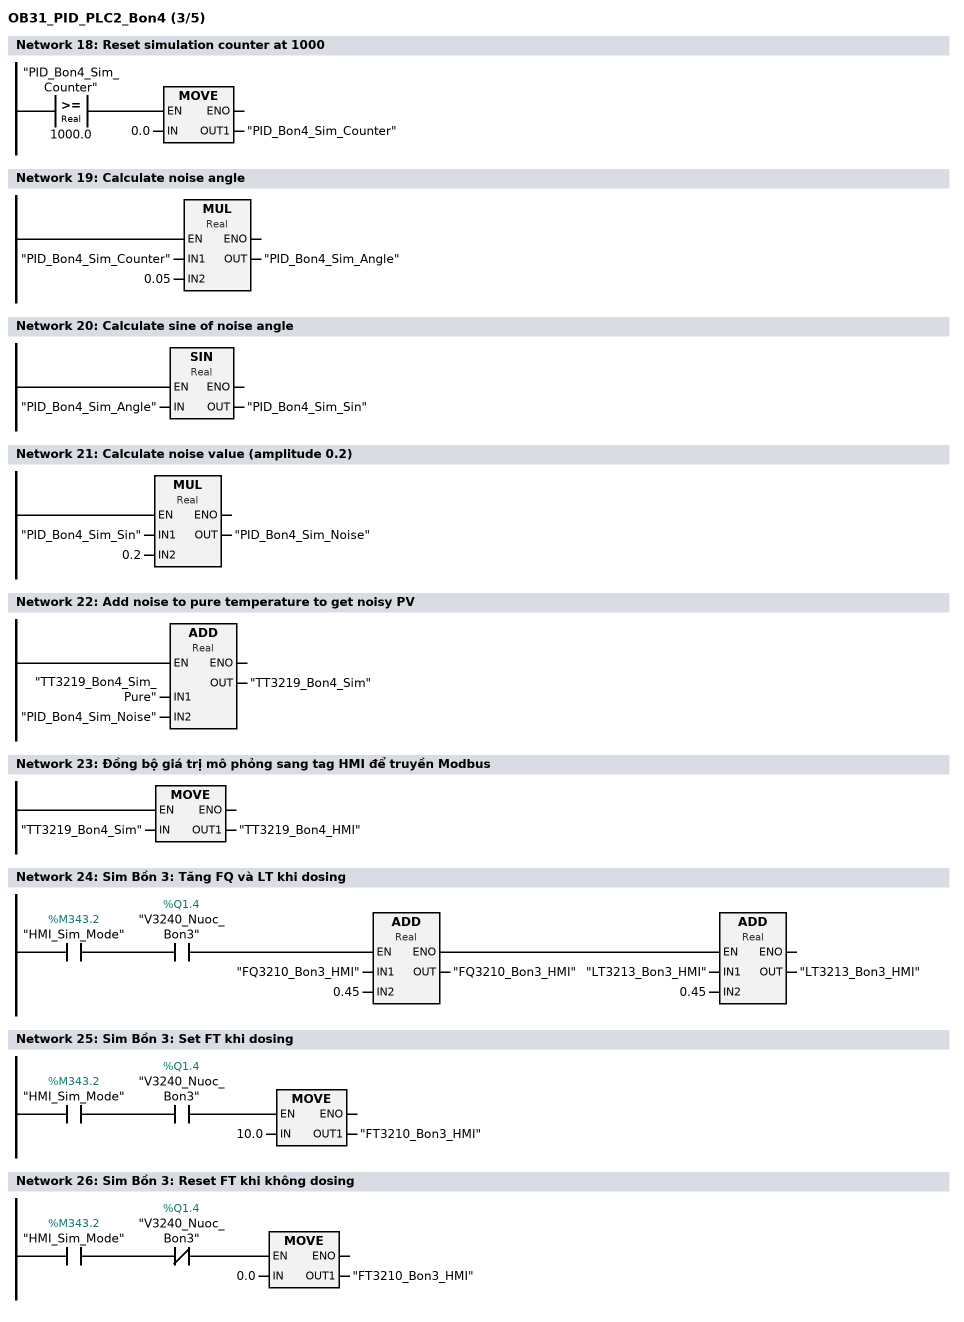
   RUNG wire#powerrail
      { S7_Templates := "SrcType := Real" } GE_Contact(in1 := "PID_Bon4_Sim_Counter", in2 := 1000.0)
      { S7_GenerateENO := "TRUE" } Move(in := 0.0, out1 => "PID_Bon4_Sim_Counter")
   END_RUNG
   // the same network as SCL:
   IF "PID_Bon4_Sim_Counter" >= 1000.0 THEN "PID_Bon4_Sim_Counter" := 0.0; END_IF;
END_REGION

REGION Network 19: Calculate noise angle
   RUNG wire#powerrail
      { S7_Templates := "SrcType := Real"; S7_GenerateENO := "TRUE" } Mul(in1 := "PID_Bon4_Sim_Counter", in2 := 0.05, out => "PID_Bon4_Sim_Angle")
   END_RUNG
   // the same network as SCL:
   "PID_Bon4_Sim_Angle" := "PID_Bon4_Sim_Counter" * 0.05;
END_REGION

REGION Network 20: Calculate sine of noise angle
   "PID_Bon4_Sim_Sin" := SIN("PID_Bon4_Sim_Angle");
END_REGION

REGION Network 21: Calculate noise value (amplitude 0.2)
   RUNG wire#powerrail
      { S7_Templates := "SrcType := Real"; S7_GenerateENO := "TRUE" } Mul(in1 := "PID_Bon4_Sim_Sin", in2 := 0.2, out => "PID_Bon4_Sim_Noise")
   END_RUNG
   // the same network as SCL:
   "PID_Bon4_Sim_Noise" := "PID_Bon4_Sim_Sin" * 0.2;
END_REGION

REGION Network 22: Add noise to pure temperature to get noisy PV
   RUNG wire#powerrail
      { S7_Templates := "SrcType := Real"; S7_GenerateENO := "TRUE" } Add(in1 := "TT3219_Bon4_Sim_Pure", in2 := "PID_Bon4_Sim_Noise", out => "TT3219_Bon4_Sim")
   END_RUNG
   // the same network as SCL:
   "TT3219_Bon4_Sim" := "TT3219_Bon4_Sim_Pure" + "PID_Bon4_Sim_Noise";
END_REGION

REGION Network 23: Đồng bộ giá trị mô phỏng sang tag HMI để truyền Modbus
   RUNG wire#powerrail
      { S7_GenerateENO := "TRUE" } Move(in := "TT3219_Bon4_Sim", out1 => "TT3219_Bon4_HMI")
   END_RUNG
   // the same network as SCL:
   "TT3219_Bon4_HMI" := "TT3219_Bon4_Sim";
END_REGION

REGION Network 24: Sim Bồn 3: Tăng FQ và LT khi dosing
   RUNG wire#powerrail
      Contact( "HMI_Sim_Mode" )
      Contact( "V3240_Nuoc_Bon3" )
      { S7_Templates := "SrcType := Real"; S7_GenerateENO := "TRUE" } Add(in1 := "FQ3210_Bon3_HMI", in2 := 0.45, out => "FQ3210_Bon3_HMI")
      { S7_Templates := "SrcType := Real"; S7_GenerateENO := "TRUE" } Add(in1 := "LT3213_Bon3_HMI", in2 := 0.45, out => "LT3213_Bon3_HMI")
   END_RUNG
   // the same network as SCL:
   // ENO of a box is taken as its EN; it also drops when the box reports an error
   IF "HMI_Sim_Mode" AND "V3240_Nuoc_Bon3" THEN
       "FQ3210_Bon3_HMI" := "FQ3210_Bon3_HMI" + 0.45;
       "LT3213_Bon3_HMI" := "LT3213_Bon3_HMI" + 0.45;
   END_IF;
END_REGION

REGION Network 25: Sim Bồn 3: Set FT khi dosing
   RUNG wire#powerrail
      Contact( "HMI_Sim_Mode" )
      Contact( "V3240_Nuoc_Bon3" )
      { S7_GenerateENO := "TRUE" } Move(in := 10.0, out1 => "FT3210_Bon3_HMI")
   END_RUNG
   // the same network as SCL:
   IF "HMI_Sim_Mode" AND "V3240_Nuoc_Bon3" THEN "FT3210_Bon3_HMI" := 10.0; END_IF;
END_REGION

REGION Network 26: Sim Bồn 3: Reset FT khi không dosing
   RUNG wire#powerrail
      Contact( "HMI_Sim_Mode" )
      I_Contact( "V3240_Nuoc_Bon3" )
      { S7_GenerateENO := "TRUE" } Move(in := 0.0, out1 => "FT3210_Bon3_HMI")
   END_RUNG
   // the same network as SCL:
   IF "HMI_Sim_Mode" AND NOT "V3240_Nuoc_Bon3" THEN "FT3210_Bon3_HMI" := 0.0; END_IF;
END_REGION

REGION Network 27: Sim Bồn 3: Giảm LT khi xả đáy
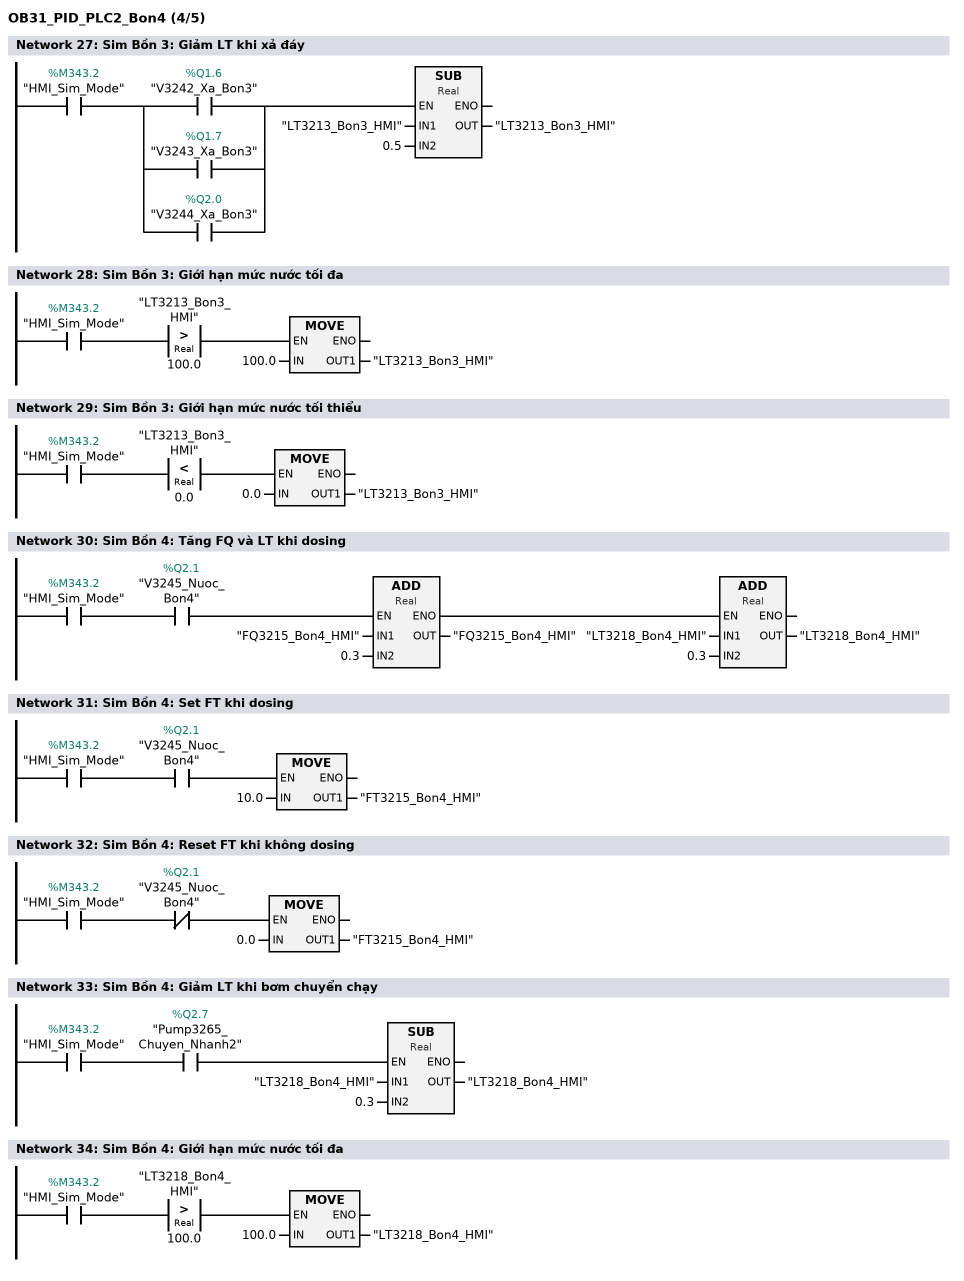
   RUNG wire#powerrail
      Contact( "HMI_Sim_Mode" )
      wire#w1
      Contact( "V3242_Xa_Bon3" )
      wire#w2
      { S7_Templates := "SrcType := Real"; S7_GenerateENO := "TRUE" } Sub(in1 := "LT3213_Bon3_HMI", in2 := 0.5, out => "LT3213_Bon3_HMI")
   END_RUNG
   RUNG wire#w1
      Contact( "V3243_Xa_Bon3" )
   END_RUNG wire#w2
   RUNG wire#w1
      Contact( "V3244_Xa_Bon3" )
   END_RUNG wire#w2
   // the same network as SCL:
   IF "HMI_Sim_Mode" AND ("V3242_Xa_Bon3" OR "V3243_Xa_Bon3" OR "V3244_Xa_Bon3") THEN
       "LT3213_Bon3_HMI" := "LT3213_Bon3_HMI" - 0.5;
   END_IF;
END_REGION

REGION Network 28: Sim Bồn 3: Giới hạn mức nước tối đa
   RUNG wire#powerrail
      Contact( "HMI_Sim_Mode" )
      { S7_Templates := "SrcType := Real" } GT_Contact(in1 := "LT3213_Bon3_HMI", in2 := 100.0)
      { S7_GenerateENO := "TRUE" } Move(in := 100.0, out1 => "LT3213_Bon3_HMI")
   END_RUNG
   // the same network as SCL:
   IF "HMI_Sim_Mode" AND ("LT3213_Bon3_HMI" > 100.0) THEN "LT3213_Bon3_HMI" := 100.0; END_IF;
END_REGION

REGION Network 29: Sim Bồn 3: Giới hạn mức nước tối thiểu
   RUNG wire#powerrail
      Contact( "HMI_Sim_Mode" )
      { S7_Templates := "SrcType := Real" } LT_Contact(in1 := "LT3213_Bon3_HMI", in2 := 0.0)
      { S7_GenerateENO := "TRUE" } Move(in := 0.0, out1 => "LT3213_Bon3_HMI")
   END_RUNG
   // the same network as SCL:
   IF "HMI_Sim_Mode" AND ("LT3213_Bon3_HMI" < 0.0) THEN "LT3213_Bon3_HMI" := 0.0; END_IF;
END_REGION

REGION Network 30: Sim Bồn 4: Tăng FQ và LT khi dosing
   RUNG wire#powerrail
      Contact( "HMI_Sim_Mode" )
      Contact( "V3245_Nuoc_Bon4" )
      { S7_Templates := "SrcType := Real"; S7_GenerateENO := "TRUE" } Add(in1 := "FQ3215_Bon4_HMI", in2 := 0.3, out => "FQ3215_Bon4_HMI")
      { S7_Templates := "SrcType := Real"; S7_GenerateENO := "TRUE" } Add(in1 := "LT3218_Bon4_HMI", in2 := 0.3, out => "LT3218_Bon4_HMI")
   END_RUNG
   // the same network as SCL:
   // ENO of a box is taken as its EN; it also drops when the box reports an error
   IF "HMI_Sim_Mode" AND "V3245_Nuoc_Bon4" THEN
       "FQ3215_Bon4_HMI" := "FQ3215_Bon4_HMI" + 0.3;
       "LT3218_Bon4_HMI" := "LT3218_Bon4_HMI" + 0.3;
   END_IF;
END_REGION

REGION Network 31: Sim Bồn 4: Set FT khi dosing
   RUNG wire#powerrail
      Contact( "HMI_Sim_Mode" )
      Contact( "V3245_Nuoc_Bon4" )
      { S7_GenerateENO := "TRUE" } Move(in := 10.0, out1 => "FT3215_Bon4_HMI")
   END_RUNG
   // the same network as SCL:
   IF "HMI_Sim_Mode" AND "V3245_Nuoc_Bon4" THEN "FT3215_Bon4_HMI" := 10.0; END_IF;
END_REGION

REGION Network 32: Sim Bồn 4: Reset FT khi không dosing
   RUNG wire#powerrail
      Contact( "HMI_Sim_Mode" )
      I_Contact( "V3245_Nuoc_Bon4" )
      { S7_GenerateENO := "TRUE" } Move(in := 0.0, out1 => "FT3215_Bon4_HMI")
   END_RUNG
   // the same network as SCL:
   IF "HMI_Sim_Mode" AND NOT "V3245_Nuoc_Bon4" THEN "FT3215_Bon4_HMI" := 0.0; END_IF;
END_REGION

REGION Network 33: Sim Bồn 4: Giảm LT khi bơm chuyển chạy
   RUNG wire#powerrail
      Contact( "HMI_Sim_Mode" )
      Contact( "Pump3265_Chuyen_Nhanh2" )
      { S7_Templates := "SrcType := Real"; S7_GenerateENO := "TRUE" } Sub(in1 := "LT3218_Bon4_HMI", in2 := 0.3, out => "LT3218_Bon4_HMI")
   END_RUNG
   // the same network as SCL:
   IF "HMI_Sim_Mode" AND "Pump3265_Chuyen_Nhanh2" THEN "LT3218_Bon4_HMI" := "LT3218_Bon4_HMI" - 0.3; END_IF;
END_REGION

REGION Network 34: Sim Bồn 4: Giới hạn mức nước tối đa
   RUNG wire#powerrail
      Contact( "HMI_Sim_Mode" )
      { S7_Templates := "SrcType := Real" } GT_Contact(in1 := "LT3218_Bon4_HMI", in2 := 100.0)
      { S7_GenerateENO := "TRUE" } Move(in := 100.0, out1 => "LT3218_Bon4_HMI")
   END_RUNG
   // the same network as SCL:
   IF "HMI_Sim_Mode" AND ("LT3218_Bon4_HMI" > 100.0) THEN "LT3218_Bon4_HMI" := 100.0; END_IF;
END_REGION

REGION Network 35: Sim Bồn 4: Giới hạn mức nước tối thiểu
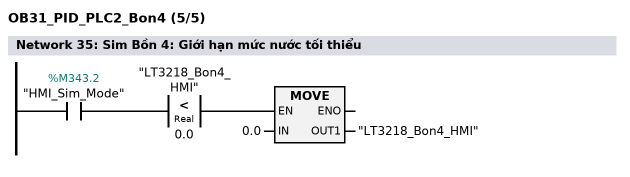
   RUNG wire#powerrail
      Contact( "HMI_Sim_Mode" )
      { S7_Templates := "SrcType := Real" } LT_Contact(in1 := "LT3218_Bon4_HMI", in2 := 0.0)
      { S7_GenerateENO := "TRUE" } Move(in := 0.0, out1 => "LT3218_Bon4_HMI")
   END_RUNG
   // the same network as SCL:
   IF "HMI_Sim_Mode" AND ("LT3218_Bon4_HMI" < 0.0) THEN "LT3218_Bon4_HMI" := 0.0; END_IF;
END_REGION
END_ORGANIZATION_BLOCK

DATA_BLOCK "MB_SERVER_DB"   // DB53
// stored: AutoNumber true, DBAccessibleFromOPCUA true, InstanceOfName MB_SERVER, OfSystemLibElement MB_SERVER, OfSystemLibVersion 3.1
"MB_SERVER"
   // VAR_INPUT
   //    DISCONNECT : Bool;
   //    CONNECT_ID : UInt;
   //    IP_PORT : UInt;
   // END_VAR
   // VAR_OUTPUT
   //    NDR : Bool;
   //    DR : Bool;
   //    ERROR : Bool;
   //    STATUS : Word;
   // END_VAR
   // VAR_IN_OUT
   //    MB_HOLD_REG : Variant;
   // END_VAR
   // VAR
   //    TCON_SFB { S7_SetPoint := 'True'} : TCON;
   //    TDISCON_SFB { S7_SetPoint := 'True'} : TDISCON;
   //    TSEND_SFB { S7_SetPoint := 'True'} : TSEND;
   //    TRCV_SFB { S7_SetPoint := 'True'} : TRCV;
   //    TCON_Param { S7_SetPoint := 'True'} : TCON_Param;
   //    MB_State : UInt;
   //    Request_Count : UInt;
   //    Server_Message_Count : UInt;
   //    Xmt_Rcv_Count : UInt;
   //    Exception_Count : UInt;
   //    Success_Count : UInt;
   //    SL_Status_Hold : UInt;
   //    HR_Start_Offset : UInt;
   //    Init_OK : Bool;
   //    SL_Error_State : Bool;
   //    Connected : Bool;
   //    XMT_Set_NDR : Bool;
   //    XMT_Set_DR : Bool;
   // END_VAR
BEGIN
   TCON_Param.CONNECTION_TYPE := 11;
   TCON_Param.LOCAL_DEVICE_ID := 64;
END_DATA_BLOCK
